// TIA Portal V17 export
// export: Created 2022-02-03T14:45:10.497602Z, ExportSetting WithDefaults, DisplayName Totally Integrated Automation Portal, DisplayVersion V17, DisplayName TIA Portal Openness, DisplayVersion V17, DisplayName TIA Portal Version Control Interface, DisplayVersion V17, DisplayName SINAMICS Startdrive Advanced, DisplayVersion V17, DisplayName SINAMICS Startdrive G130, G150, S120, S150, SINAMICS MV, S210, DisplayVersion V17, DisplayName SINAMICS Startdrive G110M, G120, G120C, G120D, G120P, G115D, DisplayVersion V17, DisplayName STEP 7 Professional, DisplayVersion V17, DisplayName STEP 7 Safety, DisplayVersion V17, DisplayName WinCC Advanced, DisplayVersion V17
FUNCTION_BLOCK "Conveyor"   // FB2, LAD
VERSION : 0.1
// stored: Access Published, AutoNumber true, IsIECCheckEnabled false, IsRetainMemResEnabled false, MemoryReserve 100, SetENOAutomatically false, UDAEnableTagReadback false
   VAR_INPUT
      operationMode : Bool;
      jogRight : Bool;
      jogLeft : Bool;
      conveyorIn : "typeConveyorInput";
      conveyorFault : Bool;
      weightOk : Bool;
      currentStoreFull : Bool;
   END_VAR
   VAR_OUTPUT
      conveyorRight : Bool;
      conveyorLeft : Bool;
   END_VAR
   VAR_IN_OUT
      occupiedBay : Array[#FIRSTBAY..#LASTBAY] of Bool;
   END_VAR
   VAR
      statAutoLeft : Bool;
      InstBayOccupied1 { S7_SetPoint := 'True'} : "BayOccupied";
      InstBayOccupied2 { S7_SetPoint := 'True'} : "BayOccupied";
      InstBayOccupied3 { S7_SetPoint := 'True'} : "BayOccupied";
   END_VAR
   VAR_TEMP
      tempManLeft : Bool;
   END_VAR
   VAR CONSTANT
      FIRSTBAY : UInt := 1;
      LASTBAY : UInt := 3;
   END_VAR
BEGIN

REGION Network 1
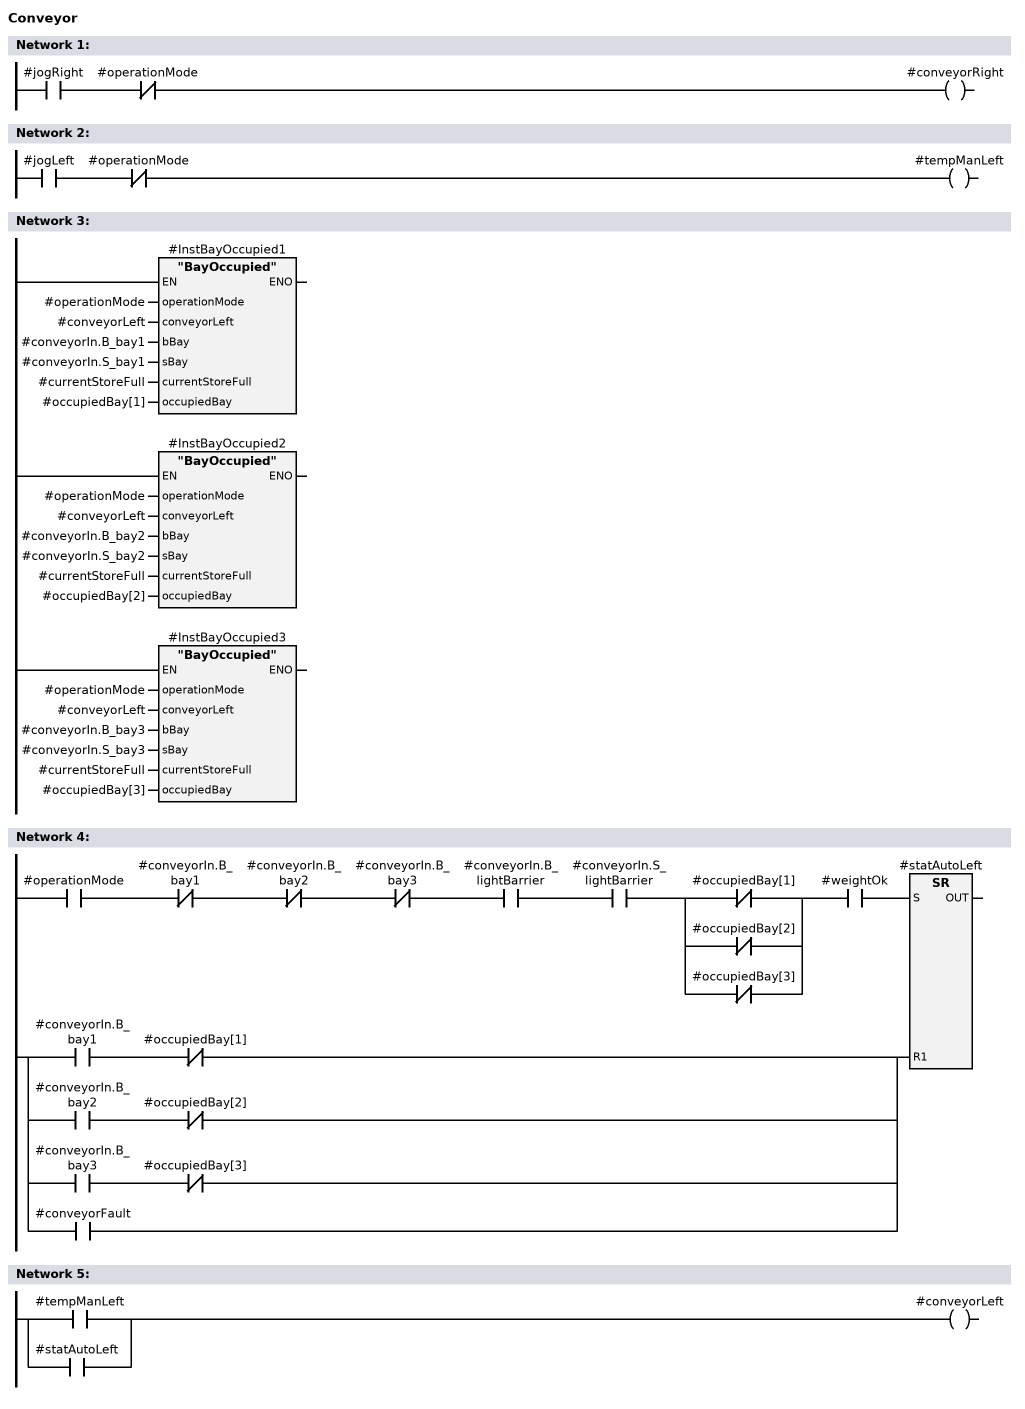
   RUNG wire#powerrail
      Contact( #jogRight )
      I_Contact( #operationMode )
      Coil( #conveyorRight )
   END_RUNG
   // the same network as SCL:
   #conveyorRight := #jogRight AND NOT #operationMode;
END_REGION

REGION Network 2
   RUNG wire#powerrail
      Contact( #jogLeft )
      I_Contact( #operationMode )
      Coil( #tempManLeft )
   END_RUNG
   // the same network as SCL:
   #tempManLeft := #jogLeft AND NOT #operationMode;
END_REGION

REGION Network 3
   RUNG wire#powerrail
      #InstBayOccupied1(operationMode := #operationMode, conveyorLeft := #conveyorLeft, bBay := #conveyorIn.B_bay1, sBay := #conveyorIn.S_bay1, currentStoreFull := #currentStoreFull, occupiedBay := #occupiedBay[1])
   END_RUNG
   RUNG wire#powerrail
      #InstBayOccupied2(operationMode := #operationMode, conveyorLeft := #conveyorLeft, bBay := #conveyorIn.B_bay2, sBay := #conveyorIn.S_bay2, currentStoreFull := #currentStoreFull, occupiedBay := #occupiedBay[2])
   END_RUNG
   RUNG wire#powerrail
      #InstBayOccupied3(operationMode := #operationMode, conveyorLeft := #conveyorLeft, bBay := #conveyorIn.B_bay3, sBay := #conveyorIn.S_bay3, currentStoreFull := #currentStoreFull, occupiedBay := #occupiedBay[3])
   END_RUNG
   // the same network as SCL:
   #InstBayOccupied1(operationMode := #operationMode,   // "BayOccupied"
                     conveyorLeft := #conveyorLeft,
                     bBay := #conveyorIn.B_bay1,
                     sBay := #conveyorIn.S_bay1,
                     currentStoreFull := #currentStoreFull,
                     occupiedBay := #occupiedBay[1]);
   #InstBayOccupied2(operationMode := #operationMode,   // "BayOccupied"
                     conveyorLeft := #conveyorLeft,
                     bBay := #conveyorIn.B_bay2,
                     sBay := #conveyorIn.S_bay2,
                     currentStoreFull := #currentStoreFull,
                     occupiedBay := #occupiedBay[2]);
   #InstBayOccupied3(operationMode := #operationMode,   // "BayOccupied"
                     conveyorLeft := #conveyorLeft,
                     bBay := #conveyorIn.B_bay3,
                     sBay := #conveyorIn.S_bay3,
                     currentStoreFull := #currentStoreFull,
                     occupiedBay := #occupiedBay[3]);
END_REGION

REGION Network 4
   RUNG wire#powerrail
      Contact( #operationMode )
      I_Contact( #conveyorIn.B_bay1 )
      I_Contact( #conveyorIn.B_bay2 )
      I_Contact( #conveyorIn.B_bay3 )
      Contact( #conveyorIn.B_lightBarrier )
      Contact( #conveyorIn.S_lightBarrier )
      wire#w1
      I_Contact( #occupiedBay[1] )
      wire#w2
      Contact( #weightOk )
      S_SR(operand := #statAutoLeft, r1 := wire#w3)
   END_RUNG
   RUNG wire#w1
      I_Contact( #occupiedBay[2] )
   END_RUNG wire#w2
   RUNG wire#w1
      I_Contact( #occupiedBay[3] )
   END_RUNG wire#w2
   RUNG wire#powerrail
      Contact( #conveyorIn.B_bay1 )
      I_Contact( #occupiedBay[1] )
   END_RUNG wire#w3
   RUNG wire#powerrail
      Contact( #conveyorIn.B_bay2 )
      I_Contact( #occupiedBay[2] )
   END_RUNG wire#w3
   RUNG wire#powerrail
      Contact( #conveyorIn.B_bay3 )
      I_Contact( #occupiedBay[3] )
   END_RUNG wire#w3
   RUNG wire#powerrail
      Contact( #conveyorFault )
   END_RUNG wire#w3
   // the same network as SCL:
   IF #operationMode AND NOT #conveyorIn.B_bay1 AND NOT #conveyorIn.B_bay2 AND NOT #conveyorIn.B_bay3 AND #conveyorIn.B_lightBarrier AND #conveyorIn.S_lightBarrier AND (NOT #occupiedBay[1] OR NOT #occupiedBay[2] OR NOT #occupiedBay[3]) AND #weightOk THEN
       #statAutoLeft := TRUE;   // SR flip-flop
   END_IF;
   IF (#conveyorIn.B_bay1 AND NOT #occupiedBay[1]) OR (#conveyorIn.B_bay2 AND NOT #occupiedBay[2]) OR (#conveyorIn.B_bay3 AND NOT #occupiedBay[3]) OR #conveyorFault THEN
       #statAutoLeft := FALSE;
   END_IF;
END_REGION

REGION Network 5
   RUNG wire#powerrail
      Contact( #tempManLeft )
      wire#w1
      Coil( #conveyorLeft )
   END_RUNG
   RUNG wire#powerrail
      Contact( #statAutoLeft )
   END_RUNG wire#w1
   // the same network as SCL:
   #conveyorLeft := #tempManLeft OR #statAutoLeft;
END_REGION
END_FUNCTION_BLOCK
